Staubli VAL3: Motion.pjx

--- Motion.pjx ---
Parameters version=s7.8.3 stackSize=5000 millimeterUnit=true
Program file=AdvanceSingal.pgx
Program file=AllMotion.pgx
Program file=chkAtHome.pgx
Program file=CloseSingnal.pgx
Program file=Control.pgx
Program file=loadPath.pgx
Program file=MainKey.pgx
Program file=Message.pgx
Program file=MotionPage.pgx
Program file=OnF1.pgx
Program file=OnF2.pgx
Program file=OnF3.pgx
Program file=OnF4.pgx
Program file=OnF5.pgx
Program file=OnF6.pgx
Program file=OnF7.pgx
Program file=OnF8.pgx
Program file=OpenSingnal.pgx
Program file=Refresh2.pgx
Program file=RefreshBelt.pgx
Program file=RefreshList.pgx
Program file=RefreshPage.pgx
Program file=sendInform.pgx
Program file=SimuMain.pgx
Program file=SingleMotion.pgx
Program file=start.pgx
Program file=StartMotion.pgx
Program file=stop.pgx
Program file=StopMotion.pgx
Program file=WholeMotion.pgx
Data file=Motion.dtx
Library alias=prd path=Disk://template/normalPath/normalPath.pjx
Library alias=PublicData path=Disk://PublicData/PublicData.pjx
Library alias=Tool path=Disk://Tool/Tool.pjx
Library alias=Frame path=Disk://Frame/Frame.pjx
Library alias=PublicProg path=Disk://PublicProg/PublicProg.pjx
Library alias=IO path=Disk://IO/IO.pjx
Library alias=SparePonit path=Disk://SparePoint/SparePoint.pjx
Library alias=user path=Disk://userPage/USERPAGE.pjx
Library alias=Pallet path=Disk://Pallet/Pallet.pjx

--- Motion.dtx ---
mdesc mNomSpeed
bool bPause
bool bRuning
bool bStop
tool tTool = {fatherId=flange[0], ioLink=valve1}
frame fFrame = {fatherId=world[0]}
pointRx pDemo = {fatherId=fFrame[0]}
string sFolder = "Disk://Traj/"
string sPtpara
configRx cConfig
num l_nRes
bool bExit
bool bUserRefresh
bool bListRefresh
string sPath
string sList
num nSelected
string sItem
string sProductList
pointRx pPoint = {fatherId=world[0]}
pointRx pSparePoint = {fatherId=world[0]}
string sMsg[8]

--- start.pgx ---
program start()
begin
  call MotionPage()
end

--- AdvanceSingal.pgx ---
program AdvanceSingal()
begin
  //需要提前开启的信号

end

--- AllMotion.pgx ---
public program AllMotion(string x_sPrd)
  local bool l_bRes
  local num l_ni
  local num l_nSize
begin
  //
  //判断安全位置
  call chkAtHome(l_bRes)
  if !l_bRes
    return
  endIf
  //
  PublicData:sStatus="stop"
  //正在加工的路径
  if PublicData:sCurrentPrd!=x_sPrd
    PublicData:sCurrentPrd=x_sPrd
    l_ni=0
    while l_ni<size(sProductList) and find(sProductList[l_ni],"P")<0
      l_ni=l_ni+1
    endWhile
    //初始化计数
    l_nSize=l_ni
    resize(PublicData:nCompenCount,1,l_nSize)
    for l_ni=0 to l_nSize-1
      PublicData:nCompenCount[l_ni]=0
    endFor
  endIf
  //
  taskCreate "control",100,Control()
  taskCreate "motion",100,WholeMotion(x_sPrd)
  call MotionPage()
end

--- chkAtHome.pgx ---
program chkAtHome(bool& x_bIsHome)
begin
  //判读机器人是否在安全位置
  if abs(PublicData:jHome)<{0.1,0.1,0.1,0.1,0.1,0.1}
    popUpMsg("机器人安全位置：6个轴都不能为零.")
    x_bIsHome=false
    return
  endIf

  if abs(herej()-PublicData:jHome)>{0.1,0.1,0.1,0.1,0.1,0.1}
    x_bIsHome=false
    popUpMsg("机器人不在安全位置。")
  else
    x_bIsHome=true
  endIf
end

--- CloseSingnal.pgx ---
program CloseSingnal()
begin
  //
  IO:dOut["dOut4"]=false
end

--- Control.pgx ---
program Control()
begin
  //
  while true
    //急停按下：结束立即结束
    if esStatus()==2
      PublicData:sStatus="Estop"
      call StopMotion()
      bExit=true
      return
    endIf
    //endstop:单循环结束停止
    if IO:diEndStop==true
      PublicData:sStatus="endstop"
      wait(IO:diEndStop==false)
    endIf

    //start/resume
    if IO:diStart==true
      //
      if PublicData:sStatus=="stop"
        PublicData:sStatus="run"
        enablePower()
      elseIf PublicData:sStatus=="pause"
        PublicData:sStatus="run"
        restartMove()
      elseIf PublicData:sStatus=="run"
        PublicData:sStatus="pause"
        stopMove()
       endIf
      wait(IO:diStart==false)
    endIf
    delay(0)
  endWhile

end

--- loadPath.pgx ---
program loadPath(bool& x_bRes, string x_sFile)
begin
  //加载路径
  x_bRes=false
  if prd:libLoad(sFolder+x_sFile)!=0
    logMsg(x_sFile+":加载失败")
    popUpMsg(x_sFile+":加载失败")
    return
  endIf
  x_bRes=true

end

--- MainKey.pgx ---
program MainKey(num x_nKey)
  local num l_nKey
begin
  //
  switch x_nKey
    //开始
    case 271
      call OnF1()
    break
    //停止
    case 272
      call OnF2()
    break
    //删除
    case 273
      call OnF3()
    break
    //编辑
    case 274
      call OnF4()
    break
    //
    case 275
    break
    //
    case 276
      call OnF6()
    break
    //save
    case 277
      call OnF7()
    break
    //返回
    case 278
      call OnF8("是否返回")
    break

  endSwitch
  wait(getKey()==-1)
end

--- Message.pgx ---
program Message(string x_sMsg, bool x_bLogShow)
  local num l_ni
begin
  //显示操作信息
  //x_sMsg:需要显示的信息
  //x_bLogShow:
  //--true:在userpage和log同时显示；
  //--false:仅在userpage中显示

  for l_ni=0 to 7
    if sMsg[l_ni]==""
      sMsg[l_ni]=x_sMsg
      l_ni=8
    elseIf l_ni==7
      for l_ni=0 to 6
        sMsg[l_ni]=sMsg[l_ni+1]
      endFor
      sMsg[l_ni]=x_sMsg
    endIf
  endFor

  for l_ni=0 to 7
    gotoxy(1,3+l_ni)
    put(sMsg[l_ni]+"     ")
  endFor
  //
  if x_bLogShow
    logMsg(sMsg)
  endIf
end

--- MotionPage.pgx ---
program MotionPage()
begin
  cls()
  bExit=false
  do
    call RefreshPage()
    call RefreshBelt()
    delay(0)
  until bExit
  bExit=false
end

--- OnF1.pgx ---
public program OnF1()
begin
  taskCreate "Motion",100,SingleMotion(sPath,true,0)
  wait(taskStatus("Motion")==1)
end

--- OnF2.pgx ---
public program OnF2()
begin
  //
  call StopMotion()
end

--- OnF3.pgx ---
public program OnF3()
begin
end

--- OnF4.pgx ---
public program OnF4()
begin
end

--- OnF5.pgx ---
public program OnF5()
begin
end

--- OnF6.pgx ---
public program OnF6()
begin
end

--- OnF7.pgx ---
public program OnF7()
begin
end

--- OnF8.pgx ---
program OnF8(string x_sMsg)
  local num l_i
  local string l_sYesNo[2]
begin
  l_sYesNo[0]="是"
  l_sYesNo[1]="否"
  call user:questionDialog(x_sMsg,l_sYesNo,l_i)
  if l_i==0 or l_i==1
    bExit=true
  endIf
  bUserRefresh=true
end

--- OpenSingnal.pgx ---
program OpenSingnal()
begin
  //外设1
  IO:dOut["dOut4"]=true
end

--- RefreshBelt.pgx ---
program RefreshBelt()
begin
  //
  gotoxy(20,1)
  put("--砂带信息--")
  gotoxy(20,3)
  put("补偿量:"+toString(".3",PublicData:nSumCompen)+"  ")
  gotoxy(20,4)
  put("补偿次数:"+toString("4",PublicData:nCompenCount)+"  ")
end

--- RefreshList.pgx ---
program RefreshList()
  local num l_ni
begin
  //


end

--- RefreshPage.pgx ---
program RefreshPage()
begin
  //
  gotoxy(1,1)
  put("--操作信息--")
//  if !bPause
//    gotoxy(1,13)
//    put("暂停")
//  else
//    gotoxy(1,13)
//    put("继续")
//  endIf

//  gotoxy(6,13)
//  put("停止")
end

--- sendInform.pgx ---
public program sendInform()
begin
  //把信号等信息传递
  //计数
  IO:dOut["dOut1"]=true
  delay(0.5)
  IO:dOut["dOut1"]=false
  //
  PublicData:nCompenCount=PublicData:nCompenCount+1
  PublicData:nSumCompen=PublicData:nCompenCount*PublicData:nDelta
  if PublicData:nCompenCount>PublicData:nBeltLife
    PublicData:nSumCompen=0
    PublicData:nCompenCount=0
    popUpMsg("更换皮带")
    stopMove()
    disablePower()
    PublicData:sStatus="pause"
    call Message("更换皮带",true)
    wait(IO:dIn["dIn1"]==true)
    call Message("皮带已更换",true)
  endIf

end

--- SimuMain.pgx ---
public program SimuMain(string x_sPath)
  local num l_nKey
begin
  //
  bExit=false
  bUserRefresh=bListRefresh=true
  sPath=x_sPath
  do
    call Refresh2()
    call RefreshList()
    call user:setList("路径",sList,bUserRefresh,bListRefresh,nSelected,sItem,l_nKey)
    bUserRefresh=false
    bListRefresh=false
    call MainKey(l_nKey)
    delay(0)
  until bExit
  bUserRefresh=bListRefresh=true
  bExit=false
end

--- SingleMotion.pgx ---
public program SingleMotion(string x_sPath, bool x_bSingle, num x_nIndex)
  local bool l_bRes
  local num l_ni
begin
  //
  call loadPath(l_bRes,x_sPath)
  if !l_bRes
    return
  endIf
  //
  //
  if x_bSingle
    tTool.trsf=prd:tTool.trsf
    fFrame.trsf=prd:fFrmMaster.trsf
  else
    //补偿
    PublicData:nSumCompen=PublicData:nCompenCount[x_nIndex]*prd:nCompDelta
    tTool.trsf=prd:tTool.trsf
    tTool.trsf.z=tTool.trsf.z-PublicData:nSumCompen
    fFrame.trsf=prd:fFrmMaster.trsf
  endIf

  //
  //
  for l_ni=0 to size(prd:pDemo)-1
    call PublicProg:SplitChar(l_nRes,prd:sPtParameter[l_ni],"/",sPtpara)
    if l_nRes<0
      return
    endIf

    //pIn
    if sPtpara[0]!="-1"
      movej(SparePonit:pPoint[sPtpara],tTool,prd:mJoint)
    endIf
    //
    if sPtpara[1]!="-1"
      movej(SparePonit:pPoint[sPtpara],tTool,prd:mJoint)
    endIf

    pDemo.trsf=prd:pDemo[l_ni].trsf
    pDemo.config=cConfig
    if l_ni==0 or l_ni==1
      movej(pDemo,tTool,prd:mJoint)
    else
      movel(pDemo,tTool,prd:mNormal)
    endIf
    //IO
    if sPtpara[3]!="-1"
      if find(sPtpara[3],"dIn")>-1
        waitEndMove()
        wait(IO:dIn[sPtpara[3]]==true)
      else
        IO:dOut[sPtpara[4]]=true
        delay(0.5)
      endIf
    endIf
    if sPtpara[4]!="-1"
      if find(sPtpara[4],"dIn")>-1
        waitEndMove()
        wait(IO:dIn[sPtpara[3]]==true)
      else
        IO:dOut[sPtpara[4]]=true
        delay(0.5)
      endIf
    endIf
    //delay
    //
    //pOut
    if sPtpara[2]!="-1"
      movej(SparePonit:pPoint[sPtpara],tTool,prd:mJoint)
    endIf

  endFor
  if x_bSingle
    waitEndMove()
  endIf

end

--- StartMotion.pgx ---
public program StartMotion(string x_sPath)
begin
  //
  taskCreate "motion",100,SingleMotion(x_sPath,true,0)
  wait(taskStatus("motion")==1)
end

--- StopMotion.pgx ---
public program StopMotion()
begin
  //
  stopMove()
  taskKill("motion")
  wait(taskStatus("motion")==-1)
  resetMotion()
  call CloseSingnal()
  PublicData:libSave()
  popUpMsg("运动结束")
end

--- WholeMotion.pgx ---
public program WholeMotion(string x_sPrdName)
  local num l_nWorkMode
  local num l_nStatus
  local bool l_bRes
  local num l_ni
  local num l_nIndex
  local num l_nj
  local num l_nk
  local num l_nCount
  local num l_nPalletCount
  local string l_sPalletName[2]
begin
  //
  while true
    l_nWorkMode=workingMode(l_nStatus)
    if PublicData:bSimulaiton
      //手动模式
      if l_nWorkMode!=1
        popUpMsg("模拟：切换到手动模式")
        wait(workingMode(l_nStatus)==1)
      endIf
    else
      //自动模式
      if l_nWorkMode!=4
        popUpMsg("生产：切换到远程模式")
        wait(workingMode(l_nStatus)==4)
      endIf
    endIf

    //判断安全位置
    call chkAtHome(l_bRes)
    if !l_bRes
      return
    endIf
    //等待启动
    call Message("等待启动",true)
    wait(IO:diStart==true)
    //机器人上电
    wait(isPowered()==true)
    call Message("运动中...",true)
    //
    //
    for l_ni=0 to size(PublicData:sPrd)-1
      if x_sPrdName==PublicData:sPrd[l_ni]
        l_nIndex=l_ni
        l_ni=size(PublicData:sPrd)+1
      endIf
    endFor

    call PublicProg:SplitChar(l_nRes,PublicData:sProductList,"/",sProductList)

    //寻找pallet的个数,最多两个pallet
    l_nPalletCount=0
    for l_ni=0 to size(sProductList)-1
      if find(sProductList[l_ni],"pallet")>-1
        l_sPalletName[l_nPalletCount]=sProductList[l_ni]
        l_nPalletCount=l_nPalletCount+1
      endIf
    endFor
    //
    call AdvanceSingal()

    //
    if l_nPalletCount==0
      //no pallet
      l_ni=0
      while find(sProductList[l_ni],"P")>-1
        if find(sProductList[l_ni+1],"P")>-1
          pSparePoint.trsf=SparePonit:pPoint[sProductList[l_ni]].trsf
          pSparePoint.config=cConfig
          movej(pSparePoint,flange,PublicData:mFast)
        else
          pSparePoint.trsf=SparePonit:pPoint[sProductList[l_ni]].trsf
          pSparePoint.config=cConfig
          movej(appro(pSparePoint,{0,0,20,0,0,0}),flange,PublicData:mFast)
          waitEndMove()
          //
          call OpenSingnal()
          movel(pSparePoint,flange,PublicData:mSlow)
          waitEndMove()
          movel(appro(pSparePoint,{0,0,20,0,0,0}),flange,PublicData:mSlow)
        endIf
        l_ni=l_ni+1
      endWhile

      //traj
      while l_ni<size(sProductList) and find(sProductList[l_ni],"P")<0

        call SingleMotion(sProductList[l_ni],false,l_ni)
        PublicData:nCompenCount[l_ni]=PublicData:nCompenCount[l_ni]+1
        l_ni=l_ni+1
      endWhile
      //

      while l_ni<size(sProductList)
        pSparePoint.trsf=SparePonit:pPoint[sProductList[l_ni]].trsf
        pSparePoint.config=cConfig
        movej(pSparePoint,flange,PublicData:mFast)
        l_ni=l_ni+1
        delay(0)
      endWhile
        waitEndMove()
      call CloseSingnal()
      movej(PublicData:jHome,flange,PublicData:mHome)
      waitEndMove()

    elseIf l_nPalletCount==1
      //one pallet
      for l_nk=0 to Pallet:uPallet[l_sPalletName[0]].ndX-1
        for l_nj=0 to Pallet:uPallet[l_sPalletName[0]].ndY-1
          //
          l_ni=0
          while find(sProductList[l_ni],"P")>-1
            pSparePoint.trsf=SparePonit:pPoint[sProductList[l_ni]].trsf
            pSparePoint.config=cConfig
            movej(pSparePoint,flange,PublicData:mFast)
            l_ni=l_ni+1
          endWhile
          //
          fFrame.trsf=Pallet:uPallet[l_sPalletName[0]].fFrame.trsf
          tTool.trsf=Tool:tTool[Pallet:uPallet[l_sPalletName[0]].sToolName].trsf
          pDemo.trsf=Pallet:uPallet[l_sPalletName[0]].pStart.trsf
          pDemo.config=cConfig
          pDemo=compose(pDemo,fFrame,{Pallet:uPallet[l_sPalletName[0]].ndX*l_nk,Pallet:uPallet[l_sPalletName[0]].ndY*l_nj,0,0,0,0})
          movej(appro(pDemo,{0,0,20,0,0,0}),tTool,PublicData:mMiddleFast)
          waitEndMove()
          //添加信号
          call OpenSingnal()
          movel(pDemo,tTool,PublicData:mSlow)
          waitEndMove()
          movel(appro(pDemo,{0,0,20,0,0,0}),tTool,PublicData:mSlow)
          //
          //traj
          while l_ni<size(sProductList) and find(sProductList[l_ni],"P")<0
            //
            call SingleMotion(sProductList[l_ni],false,l_ni)
            l_ni=l_ni+1
          endWhile

          while l_ni<size(sProductList)
            pSparePoint.trsf=SparePonit:pPoint[sProductList[l_ni]].trsf
            pSparePoint.config=cConfig
            movej(pSparePoint,flange,PublicData:mFast)
            l_ni=l_ni+1
            delay(0)
          endWhile
          waitEndMove()
          call CloseSingnal()
          movej(PublicData:jHome,flange,PublicData:mHome)
          waitEndMove()
        endFor
      endFor
    elseIf l_nPalletCount==2
      //two pallet
    endIf
    if PublicData:sStatus=="endstop"
      disablePower()
    endIf
    PublicData:sStatus="stop"
    delay(0)
  endWhile
end
